(* PLC project Generated.project, CODESYS CODESYS V3.5 SP19 Patch 1 *)
(* stored: creationDateTime 2026-09-01T01:00:13.859519, modificationDateTime 2026-09-01T01:00:13.859519 *)

(* ═══════════════════════════════════════════════════════════════ ⚙️ ST_CycleDumpAtTremieCfg — Réglages persistants cycle vidage trémie (legacy) ═══════════════════════════════════════════════════════════════ *)
TYPE ST_CycleDumpAtTremieCfg : STRUCT
  Initialized : BOOL := FALSE;  (* 🚦 flag restauration boot *)
END_STRUCT;
END_TYPE

(* ======================================================================= 💾 FB_CfgPersistBridge_CycleDumpAtTremieCfg — Pont persistance cycle vidage trémie ─────────────────────────────────────────────────────────────── 🎯 Rôle : Restauration et synchronisation bidirectionnelle IHM / Persist 💾 Persistance : Transfert GVL_PERSISTENT <-> GVL_IHM sur Initialized 📄 Doc métier : DOC/AF/AF_Partie-03_Contrats_Composants_v2.3.md §3 ======================================================================= *)
FUNCTION_BLOCK FB_CfgPersistBridge_CycleDumpAtTremieCfg
  VAR_OUTPUT
    JustRestored : BOOL;  (* === ETATS RESTAURATION === <-- [STAT] Vrai sur le cycle de restauration initiale *)
  END_VAR
  VAR_IN_OUT
    Hmi : ST_CycleDumpAtTremieCfg;  (* === BUS CONFIGURATION ET PERSISTANCE === <-> [BUS] Structure de configuration IHM *)
    Persist : ST_CycleDumpAtTremieCfg;  (* <-> [BUS] Structure de configuration persistante *)
  END_VAR

            

JustRestored := FALSE;
IF NOT Hmi.Initialized THEN
    Hmi := Persist;
    Hmi.Initialized := TRUE;
    JustRestored := TRUE;
ELSE
    Persist := Hmi;
END_IF;

          
END_FUNCTION_BLOCK
